Staubli VAL3: SETLIST.pgx

public program setList(string x_sTitle, string& x_sListItem[], bool x_bUserRefresh, bool x_bListItemRef, num& x_nSelected, string& x_sItem, num& x_nKey)
  local num l_nView
  local num l_nItem
begin
  if x_bUserRefresh
    if x_bListItemRef
      call setSizeList(20,0,18,11)
      call listcreate(x_sTitle)
      if x_sListItem[0]!=""
        call listadd(x_sListItem)
      endIf
    else
      call setSizeList(20,0,18,11)
      call listframe(x_sTitle,nTopX,nTopY,nBottomX,nBottomY)
    endIf
    call selectNewField(x_nSelected,l_nItem,l_nView)
  endIf
  x_nKey=getKey()
  if x_nKey!=-1
    call listevent(x_nKey,l_nItem,x_sItem)
    l_nView=nView
    x_nSelected=l_nItem
  endIf
end
